TYPE EtcSlaveBase_82538BE2 :
STRUCT
END_STRUCT
END_TYPE

(* stored: Version 1.2.0.0, ProductVersion 3.1.4024.9
   DUT EtcSlaveBase_82538BE2: Id {3f2f6888-caba-4fdb-88af-431faa3d1d71} *)
